// TIA Portal V17 export
// export: Created 2024-09-02T12:50:05.1808032Z, ExportSetting WithDefaults, DisplayName Totally Integrated Automation Portal, DisplayVersion V17, DisplayName TIA Portal Openness, DisplayVersion V17, DisplayName TIA Portal Version Control Interface, DisplayVersion V17, DisplayName STEP 7 Professional, DisplayVersion V17, DisplayName STEP 7 Safety, DisplayVersion V17, DisplayName WinCC Professional, DisplayVersion V17
FUNCTION_BLOCK "CPU Monitoring"   // FB4, LAD
{ S7_Optimized_Access := 'TRUE' }
VERSION : 0.1
// stored: AutoNumber true, IsIECCheckEnabled false, IsRetainMemResEnabled false, MemoryReserve 100, SetENOAutomatically false, UDAEnableTagReadback false
   VAR
      Mode : UInt := 11;
      OBnr : OB_ANY := 1001;
      InfoData : UInt;
      ReturnValue : Int;
   END_VAR
BEGIN

REGION Network 1
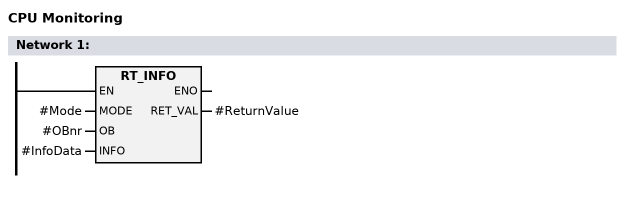
   RUNG wire#powerrail
      RT_INFO(MODE := #Mode, OB := #OBnr, INFO := #InfoData, Ret_Val => #ReturnValue)
   END_RUNG
   // the same network as SCL:
   #ReturnValue := RT_INFO(MODE := #Mode, OB := #OBnr, INFO := #InfoData);
END_REGION
END_FUNCTION_BLOCK
